FUNCTION_BLOCK FB_Tote_Subsystem
VAR_INPUT
END_VAR
VAR_OUTPUT
END_VAR
VAR
	status	: MachineStatus := MachineStatus.STOPPED;	
	current_air_pressure	: REAL;	
	machine_control_cmd	: MachineControlCommand;

	ton1	: TON;

	ton_heart_beat	: TON;
	bReset_ads_heart_beat	: BOOL;
	bTest	:BOOL;
	
	machine_current_status	: E_PMLState;


END_VAR

M_mapping();

machine_current_status	:= GVL.PackTags.Status.StateCurrent;

CASE machine_current_status OF
	ePMLState_Aborted,ePMLState_Aborting:
		status	:= MachineStatus.ERROR;
	ePMLState_Stopping:	
		status	:= MachineStatus.STOPPING;
	ePMLState_Stopped:
		status	:= MachineStatus.STOPPED;
	ePMLState_Resetting:	
		status	:= MachineStatus.RESETTING;
	ePMLState_Idle:	
		status	:= MachineStatus.READY;		
	ePMLState_Execute:	
		status	:= MachineStatus.RUNNING;			
		
END_CASE




/////////////////////////test/////////////////
ton1(PT:=T#1S);
IF bTest THEN//test ads heart beat
	ads_heart_beat(i:=1);
	bTest	:= FALSE;
END_IF
//////////////////////////ads heart beat/////////////////
ton_heart_beat(IN:=NOT bReset_ads_heart_beat,PT:=T#3S);
IF bReset_ads_heart_beat THEN
	bReset_ads_heart_beat	:= FALSE;
END_IF

{attribute 'TcRpcEnable'}
METHOD ads_heart_beat : BOOL
VAR_INPUT
	i	: INT;
END_VAR
ads_heart_beat	:= FALSE; 
bReset_ads_heart_beat	:= TRUE;
ads_heart_beat	:= TRUE;
END_METHOD

METHOD M_mapping : BOOL
VAR_INPUT
END_VAR
END_METHOD

{attribute 'TcRpcEnable'}
METHOD machine_control_command : BOOL
VAR_INPUT
	Command	: MachineControlCommand;
END_VAR
machine_control_command	:= FALSE; 

machine_control_cmd	:= Command;

machine_control_command	:= TRUE;
END_METHOD

END_FUNCTION_BLOCK

(* stored: Version 1.1.0.1, ProductVersion 3.1.4024.12
   POU FB_Tote_Subsystem: Id {18f3e813-8d9e-4f02-997f-31b8e26895c7}, SpecialFunc None
   Method ads_heart_beat: Id {fd3aacdd-bd79-468f-b337-c73a0025f4da}
   Method M_mapping: Id {541fb1a0-cd7a-4efb-8c21-3483a35c300d}
   Method machine_control_command: Id {e35d6b29-fce8-4046-8fa5-9d1764fae381} *)
